PROGRAM POU
VAR
END_VAR

// NETWORK 1

END_PROGRAM

(* stored: Version 1.1.0.1, ProductVersion 3.1.4024.12
   POU POU: Id {836f32ed-eb68-4810-b301-3c8dcf604713}, SpecialFunc None *)
